FUNCTION_BLOCK FB_AutoPlace
VAR_INPUT
	BlueStopper : BOOL;
	
END_VAR
VAR_OUTPUT
	Reader_Trigger : BOOL;
END_VAR
VAR
	Cont_Timer : ton;
	last_triggered: BOOL;
	start: BOOL;
END_VAR


Cont_Timer(IN:= BlueStopper, PT:= T#3S, Q=> , ET=> );
IF BlueStopper AND Cont_Timer.Q THEN
	//
	Reader_Trigger := TRUE;
ELSE 
	//
	Reader_Trigger := FALSE;
END_IF

//last_triggered := BlueStopper;

END_FUNCTION_BLOCK

(* stored: Version 1.1.0.1, ProductVersion 3.1.4024.12
   POU FB_AutoPlace: Id {8f407f19-b82e-4e02-897c-85d6d44e4f47}, SpecialFunc None *)
